// TIA Portal V17 export
// export: Created 2026-01-01T00:00:00, ExportSetting WithDefaults, DisplayName synthetic-fixture, DisplayVersion machine-intelligence-v1.0.0
DATA_BLOCK "DB_Line"   // DB
BEGIN
END_DATA_BLOCK
